(*
 receive a request : source on destination
 calculate the  path
 verify required resources
 reserve the relevant Ltu or conveyors
 give a ST_Route to the route executor
*)

FUNCTION_BLOCK FB_RouteManagerDevice EXTENDS FD_Device 
VAR_INPUT
END_VAR

VAR_OUTPUT
END_VAR

VAR
	//===================== interface
 	itfLTU3  											: ITF_LTU;
 	itfLTU6  											: ITF_LTU;
 	itfLTU9  											: ITF_LTU;
 	itfLTU12 											: ITF_LTU;
          											
	itfC3    											: ITF_Convoyer;
	itfC6    											: ITF_Convoyer;
	itfC9    											: ITF_Convoyer;
	itfC12   											: ITF_Convoyer;
	
	//===================== Variable
	eSource			 									: E_Convoyer;
	eDestination 									: E_Convoyer;
	
	bRouteRequest   							: BOOL;
	bRouteAvailable 							: BOOL;
  bRouteReserved								: BOOL;
	
	//===================== Instance
	
																							
END_VAR

VAR CONSTANT
	// --------------------------Base------------------
	C_SeqStep_OnBasePos_Start								: UINT :=  10; 
	C_SeqStep_OnBasePos_Wait      					: UINT :=  30;
	C_SeqStep_OnBasePos_Done								: UINT :=  40; 
	
	// --------------------------Auto Sequence---------
	C_SeqStep_Auto_Start										: UINT :=  100;
	C_SeqStep_Auto_End											: UINT :=  200;
END_VAR


//******* Important and necessary
SUPER^();  
//====================================
IF NOT Enable THEN RETURN; END_IF

PROPERTY CarrierPresent : BOOL
GET
CarrierPresent := bCarrierPresent;
END_GET
SET
bCarrierPresent := CarrierPresent;
END_SET
END_PROPERTY

//FB_Init ist immer implizit verfügbar und wird primär für die Initialisierung verwendet.
//Der Rückgabewert wird nicht ausgewertet. Für gezielte Einflussnahme können Sie
//die Methoden explizit deklarieren und darin mit dem Standard-Initialisierungscode 
//zusätzlichen Code bereitstellen. Sie können den Rückgabewert auswerten.
METHOD FB_Init: BOOL
VAR_INPUT    
	bInitRetains					: BOOL; 					// TRUE: Die Retain-Variablen werden initialisiert (Reset warm / Reset kalt)    
	bInCopyCode						: BOOL;  					// TRUE: Die Instanz wird danach in den Kopiercode kopiert (Online-Change)
	
	I_Name                : STRING;         //  Name
	I_ID                  : UINT;           // ID
  I_itfOwner					  : ITF_Owner;      // owner 
END_VAR
END_METHOD

PROPERTY LTUFree : BOOL
GET

LTUFree := bLTUFree;
END_GET
SET
bLTUFree := LTUFree;
END_SET
END_PROPERTY

PROPERTY LTUPosition : E_LTUPosition
GET
LTUPosition := eLTUPosition;
END_GET
SET
eLTUPosition := LTUPosition;
END_SET
END_PROPERTY

METHOD mAutomatic : E_CmdState
VAR_INPUT
	I_bExecute	: BOOL;
END_VAR
END_METHOD

METHOD mBuildRoute : BOOL
VAR_INPUT
	
END_VAR
// No command requested.
END_METHOD

METHOD mCheckRouteFree : BOOL
VAR_INPUT
	
END_VAR
// No command requested.
END_METHOD

METHOD mCmdExec_Auto : E_CmdState
VAR_INPUT
END_VAR

CASE SequenceID OF

  //******************************************************* Idle 
  C_SeqStep_Idle: 
  	SequenceID       :=  C_SeqStep_OnBasePos_Start;
  
  //****************************************************** Start
  C_SeqStep_OnBasePos_Start:
  	
  	SequenceID       :=  C_SeqStep_OnBasePos_Start;
	
  C_SeqStep_Error: 
    //************* all FB reset

		//************* 
  	
 	C_SeqStep_OnBasePos_Done:
  	mCmdExec_Auto := mDone();

END_CASE
END_METHOD

METHOD mCmdExec_BasePos : E_CmdState
VAR_INPUT
END_VAR

CASE SequenceID OF

  //******************************************************* Idle 
  C_SeqStep_Idle: 
  	SequenceID       :=  C_SeqStep_Start;
  
  //****************************************************** Start
  C_SeqStep_Start:
	//
	Homed := TRUE;
  Ready := TRUE;
  SequenceID := C_SeqStep_OnBasePos_Done;
	
  C_SeqStep_Error: 
    //************* all FB reset
    mCmdExec_BasePos := mDone(); 
  //**********************Done
 	C_SeqStep_OnBasePos_Done:
  	mCmdExec_BasePos := mDone();

END_CASE
END_METHOD

METHOD mCmdExec_Service : E_CmdState
VAR_INPUT
END_VAR
;
END_METHOD

METHOD mHold : E_CmdState
VAR_INPUT
	I_bExecute	: BOOL;
END_VAR

SUPER^.mHold(I_bExecute);
END_METHOD

METHOD mHome : E_CmdState
VAR_INPUT
	I_bExecute	: BOOL;
END_VAR

SUPER^.mHome(I_bExecute);
END_METHOD

METHOD mRelease : E_CmdState
VAR_INPUT
	I_bExecute	: BOOL;
END_VAR

SUPER^.mRelease(I_bExecute);
END_METHOD

METHOD mRequestRoute : E_CmdState
VAR_INPUT
   I_bExecute     		: BOOL;
   I_eSource      		: E_Convoyer;
   I_eDestination 		: E_Convoyer;
END_VAR

VAR
	L_eCmdState 					: E_CmdState;
END_VAR
// No command requested.
IF NOT I_bExecute 
	THEN
  	mRequestRoute 			:= E_CmdState.Idle;
    RETURN;         		
END_IF              		
                    		
eSource 								:= I_eSource;
eDestination 					  := I_eDestination;

IF eSource = E_Convoyer.Convoyer_NONE OR 
	 eDestination = E_Convoyer.Convoyer_NONE 
	 	THEN
    	mRequestRoute     := E_CmdState.Error;
    	RETURN;
END_IF

IF NOT mBuildRoute() 
	THEN
    mRequestRoute       := E_CmdState.Error;
    RETURN;
END_IF

IF NOT mCheckRouteFree() 
	THEN
    mRequestRoute 			:= E_CmdState.NotReady;
    RETURN;
END_IF

IF NOT mReserveRoute() 
	THEN
    mRequestRoute 			:= E_CmdState.NotReady;
    RETURN;
END_IF

bRouteAvailable 				:= TRUE;
bRouteReserved 					:= TRUE;

mRequestRoute 					:= E_CmdState.Succeeded;
END_METHOD

METHOD mReserveRoute : BOOL
VAR_INPUT
	
END_VAR
// No command requested.
END_METHOD

METHOD mSequence : E_CmdState
VAR_INPUT
	I_bExecute				: BOOL;
END_VAR

VAR_INST
	L_eCmdState 		 : E_CmdState; // To Generic checks from parent state 
	
END_VAR
mSequence := SUPER^.mSequence(I_bExecute);	


// Generic checks from parent
L_eCmdState := SUPER^.mSequence(I_bExecute := I_bExecute);

IF L_eCmdState <> E_CmdState.Busy 
	THEN
    mSequence := L_eCmdState;
    RETURN;
END_IF

CASE Mode OF
	E_Mode.Homing:
		mSequence := mCmdExec_BasePos();		
	E_Mode.Auto:
		mSequence := mCmdExec_Auto();	
	E_Mode.Service:
		mSequence := mCmdExec_Service();	
END_CASE
END_METHOD

METHOD mService : E_CmdState
VAR_INPUT
	I_bExecute	: BOOL;
END_VAR

SUPER^.mService(I_bExecute);
END_METHOD

METHOD mStop : E_CmdState
VAR_INPUT
	I_bExecute	: BOOL;
END_VAR

SUPER^.mStop(I_bExecute);
END_METHOD

PROPERTY ReservedBy : E_Convoyer
GET
ReservedBy := eReservedBy;
END_GET
SET
eReservedBy := ReservedBy;
END_SET
END_PROPERTY

END_FUNCTION_BLOCK

(* stored: Version 1.1.0.1, ProductVersion 3.1.4026.18
   POU FB_RouteManagerDevice: Id {8270a267-7ccc-4c56-898e-a1440cf6b64c}, SpecialFunc None
   Folder 01 Properties: Id {85cf6baa-21e4-4eab-a250-484e0149eff4}
   Folder 02 Methodes: Id {7ada561f-4a10-4dab-8217-abe504d828f1}
   Folder 100 CmdExecute: Id {0313f81c-d9a9-4b37-95e5-806775012e03}
   Property CarrierPresent: Id {28a673b2-92d9-4578-9add-5105e9b22dff}
   Get Get: Id {cd977f3d-1cc9-4142-82f8-0df85badda43}
   Set Set: Id {01e77b4c-da8f-432e-a40e-1981853395ff}
   Method FB_Init: Id {f025e0f4-08c7-4495-afa3-601541f6e854}
   Property LTUFree: Id {49fa8a07-b1e5-48b2-90fe-944d56de56a3}
   Get Get: Id {aba29ed6-c00d-4836-a0ff-b45e09ae0b67}
   Set Set: Id {da6fa49d-0e20-4c3d-9bef-f3d9525c3bf6}
   Property LTUPosition: Id {8f4bacc7-bc81-4d32-a31f-03cc1155a60b}
   Get Get: Id {f1c87639-7def-4256-904d-e18349e053ea}
   Set Set: Id {8871ae61-30fb-4d1c-9a4f-2f686729bd3b}
   Method mAutomatic: Id {96a825f9-7aeb-41cb-a336-78f3a907220b}
   Method mBuildRoute: Id {7200bf03-7fa0-4280-a8ff-c4a05727f4d4}
   Method mCheckRouteFree: Id {677ed7d3-36c4-4960-8f5d-5f1bc61e49dd}
   Method mCmdExec_Auto: Id {8119614c-5c76-4267-a8ee-e2944e67878d}
   Method mCmdExec_BasePos: Id {d65780c7-4e9f-42a3-9358-58c323439d29}
   Method mCmdExec_Service: Id {f8896431-6abb-450c-98ff-dfb8e5b37029}
   Method mHold: Id {fb155185-5dd5-45a4-8ccd-2c88c48f99cd}
   Method mHome: Id {70f1a819-da67-4528-b36e-9effb9c23247}
   Method mRelease: Id {9fc9f7cd-d81c-45c4-94fb-80fa991ddff3}
   Method mRequestRoute: Id {4a417486-f8d2-4dd6-9779-5933800df322}
   Method mReserveRoute: Id {b2fe83f5-9021-4c29-a99a-0b7e44acec3e}
   Method mSequence: Id {9d46ef71-25fa-47b2-8325-82cf496e3abc}
   Method mService: Id {aa5a7582-2696-4d03-8fdd-0d09e4564bca}
   Method mStop: Id {f5b09365-1a2f-4597-adcb-e0c7898af24e}
   Property ReservedBy: Id {4be86b5b-4bbe-4304-abbc-ee6242639d87}
   Get Get: Id {ee9999dc-ecd5-48f5-a251-e105ba0d0c1f}
   Set Set: Id {ec09d9d5-f6e3-4d28-9036-78bfd4186a9e} *)
